// TIA Portal V20 export
DATA_BLOCK "F-DB_DigitalInputs"   // DB110, F_DB
// stored: AutoNumber false, InstanceOfName F-FB_DigitalInput, InstanceOfType FB
"F-FB_DigitalInput"
   // VAR
   //    sSafety_EStop : EV1oo2DI;
   //    sKeySettingMode : EV1oo2DI;
   //    sKeySettingLaser : EV1oo2DI;
   //    sMaintenanceDoorClosed : EV1oo2DI;
   //    sFrontDoorClosed : EV1oo2DI;
   //    sEmergencyStopPowerLaser : EV1oo2DI;
   //    sRoofLeftDoorClosed : EV1oo2DI;
   //    sKeyLaserON : EV1oo2DI;
   //    sLaserExternDoorClosed : EV1oo2DI;
   //    sSasOneDoorClosed : EV1oo2DI;
   //    sBwLoaderDoorClosed : EV1oo2DI;
   //    sRoofRightDoorClosed : EV1oo2DI;
   //    sSonplas_EStop : EV1oo2DI;
   //    sBwLoader_EStop : EV1oo2DI;
   //    sSonplasDoorClosed : EV1oo2DI;
   //    sAck_iSafety_EStop { ExternalAccessible := 'False'; ExternalVisible := 'False'; ExternalWritable := 'False'} : Bool;
   //    sAck_iKeySettingMode { ExternalAccessible := 'False'; ExternalVisible := 'False'; ExternalWritable := 'False'} : Bool;
   //    sAck_iKeySettingLaser { ExternalAccessible := 'False'; ExternalVisible := 'False'; ExternalWritable := 'False'} : Bool;
   //    sAck_iMaintenanceDoorClosed { ExternalAccessible := 'False'; ExternalVisible := 'False'; ExternalWritable := 'False'} : Bool;
   //    sAck_iFrontDoorClosed { ExternalAccessible := 'False'; ExternalVisible := 'False'; ExternalWritable := 'False'} : Bool;
   //    sAck_iEmergencyStopPowerLaser { ExternalAccessible := 'False'; ExternalVisible := 'False'; ExternalWritable := 'False'} : Bool;
   //    sAck_iRoofLeftDoorClosed { ExternalAccessible := 'False'; ExternalVisible := 'False'; ExternalWritable := 'False'} : Bool;
   //    sAck_iKeyLaserON { ExternalAccessible := 'False'; ExternalVisible := 'False'; ExternalWritable := 'False'} : Bool;
   //    sAck_iLaserExternDoorClosed : Bool;
   //    sAck_iSasOneDoorClosed { ExternalAccessible := 'False'; ExternalVisible := 'False'; ExternalWritable := 'False'} : Bool;
   //    sAck_iBwLoaderDoorClosed : Bool;
   //    sAck_iRoofRightDoorClosed { ExternalAccessible := 'False'; ExternalVisible := 'False'; ExternalWritable := 'False'} : Bool;
   //    sAck_iSonplas_EStop : Bool;
   //    sAck_iBwLoader_EStop : Bool;
   //    sAck_iSonplasDoorClosed { ExternalAccessible := 'False'; ExternalVisible := 'False'; ExternalWritable := 'False'} : Bool;
   // END_VAR
BEGIN
END_DATA_BLOCK
